(* PLC project LdDemo, ACME plc-programming plugin 1.0 *)
(* stored: creationDateTime 2026-01-01T00:00:00 *)

PROGRAM LatchMotor
  VAR
    Start : BOOL;
    Stop : BOOL;
    Motor : BOOL;
  END_VAR
  VAR  (* added by the conversion: wires and edge detectors of the diagram *)
    R_TRIG1 : R_TRIG;
  END_VAR

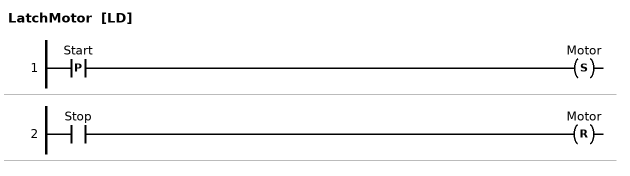
(* LD diagram, written out as Structured Text *)
R_TRIG1(CLK := Start);
IF R_TRIG1.Q THEN Motor := TRUE; END_IF;
IF Stop THEN Motor := FALSE; END_IF;
END_PROGRAM
